FUNCTION_BLOCK C_HTTP_REQUEST EXTENDS C_HTTP_BASE
VAR_INPUT
END_VAR
VAR_OUTPUT
END_VAR
VAR
	_MethodRequest		: E_HTTP_VERBS;
	_Url				: STRING(255);	
	_c_HttpVersion 		: C_HTTP_VERSION(Major_Version:= 1, Minor_Version:= 1);
	
	_Header 			: ARRAY[0..15] OF C_HTTP_HEADER(Name:= '');
	
	_MessageBody		: T_HTTPSTRING;
END_VAR

METHOD PRIVATE Get_Headers : STRING(255)
VAR_INPUT
END_VAR
VAR 
	_m : INT := 0;
	_mn : INT := 15;
	_buffer : STRING(255) := '';
END_VAR
FOR _m := 0 TO _mn BY 1 DO
	_buffer := CONCAT(_buffer, THIS^._Header[_m].ToString());
END_FOR
Get_Headers := _buffer;
END_METHOD

METHOD PRIVATE Get_RequestLine : String(255)
VAR_INPUT
END_VAR
Get_RequestLine :=	CONCAT(LV2_HTTP_DATA_DEFINITIONS.HTTP_VERB_STRING[THIS^._MethodRequest],
						CONCAT(SUPER^.Line_Space, 
							CONCAT(_Url,
								CONCAT(SUPER^.Line_Space,
									CONCAT(_c_HttpVersion.ToString(),
										SUPER^.Line_Terminator
									)
								)
							)
						)
					);
END_METHOD

PROPERTY Major_Version : uint
GET
Major_Version := _c_HttpVersion.Major;;
END_GET
END_PROPERTY

PROPERTY Message_Body : STRING(255)
GET
Message_Body := _MessageBody;
END_GET
SET
_MessageBody := Message_Body;
END_SET
END_PROPERTY

PROPERTY Minor_Version : uint
GET
Minor_Version := _c_HttpVersion.Minor;
END_GET
END_PROPERTY

METHOD Parse : RETURN_CODE
VAR_INPUT
END_VAR
END_METHOD

METHOD ToString : STRING(255)
VAR_INPUT
END_VAR
ToString :=	CONCAT(THIS^.Get_RequestLine(),
				CONCAT(THIS^.Get_Headers(),
					CONCAT(SUPER^.Line_Terminator,
						THIS^.Message_Body
					)
				)
			);
END_METHOD

PROPERTY Url : String(255)
GET
Url := _url;
END_GET
SET
_url := url;
END_SET
END_PROPERTY

PROPERTY Verb : E_HTTP_VERBS
GET
Verb := _MethodRequest;
END_GET
SET
_MethodRequest := Verb;
END_SET
END_PROPERTY

END_FUNCTION_BLOCK

(* stored: Version 1.1.0.1, ProductVersion 3.1.4019.2
   POU C_HTTP_REQUEST: Id {5aaf8f33-78a8-41e3-a1f3-83656888a26d}, SpecialFunc None
   Folder Methods: Id {9321cddf-9f72-48f7-b1a7-a80432ca3e2b}
   Folder Properties: Id {922f8cdd-ac87-4267-9d42-e1bb879e8e7a}
   Folder Internal: Id {76de9fbd-2f27-4ba5-a021-aa0e2becb3c7}
   Folder Version: Id {dcd97dd3-f8e3-4dd8-9437-8284b1479537}
   Method Get_Headers: Id {27d98323-943a-4ceb-b1d6-9c47468ef749}
   Method Get_RequestLine: Id {00a47902-09f4-4462-9b62-6a478b36dffd}
   Property Major_Version: Id {5d4b69ce-8362-49f8-b4b0-9869e8918a1f}
   Get Get: Id {b39c4944-3f87-4491-9fed-53d0e3fd9ec0}
   Property Message_Body: Id {f72234e5-ba85-4c9a-b5ec-f1596c8f1ee1}
   Get Get: Id {af83e74c-6790-4075-ae31-2ac30567af4c}
   Set Set: Id {8a71a302-29f5-4d39-8cea-5935f366f4f8}
   Property Minor_Version: Id {56fb7b69-3012-4101-b607-2307b2a51d27}
   Get Get: Id {605269c8-09de-434e-ad6f-76adad33e88c}
   Method Parse: Id {01eb5aa1-30a9-4a5f-bcf1-bfa7d86f8816}
   Method ToString: Id {761de4c4-a5c1-4c6f-b3e9-de8958253803}
   Property Url: Id {578780b4-7864-4a36-8c28-da2e47140761}
   Get Get: Id {9b00c056-496a-4b4f-b1c7-c1b12e94dfa8}
   Set Set: Id {22c218c2-baa9-4c3c-87a5-e310905332d7}
   Property Verb: Id {543ae445-cb7f-4c06-b539-f01e21b8cdda}
   Get Get: Id {55de2d47-f084-4991-ad81-40e8be6663e5}
   Set Set: Id {1c2d1c25-2220-46da-b634-753fd8aca037} *)
